// TIA Portal V18 export
// export: Created 2026-03-12T16:04:36.0251046Z, ExportSetting WithDefaults, DisplayName Totally Integrated Automation Portal, DisplayVersion V18 Update 5, DisplayName TIA Portal Openness, DisplayVersion V18 Update 5, DisplayName TIA Portal Version Control Interface, DisplayVersion V18, DisplayName SINAMICS Startdrive Advanced, DisplayVersion V18, DisplayName SINAMICS Startdrive G130, G150, S120, S150, SINAMICS MV, S210, DisplayVersion V18, DisplayName SINAMICS Startdrive G110M, G120, G120C, G120D, G120P, G115D, DisplayVersion V18, DisplayName STEP 7 Professional, DisplayVersion V18 Update 5, DisplayName STEP 7 Safety, DisplayVersion V18, DisplayName WinCC Professional, DisplayVersion V18 Update 5
FUNCTION_BLOCK "FB_MOVE_SKID_UV"   // FB40, LAD
{ S7_Optimized_Access := 'TRUE' }
VERSION : 0.1
// stored: AutoNumber true, IsIECCheckEnabled false, IsRetainMemResEnabled false, MemoryReserve 100, SetENOAutomatically false, UDAEnableTagReadback false
   VAR_INPUT
      UV_IN : Array[0..4] of Byte;
   END_VAR
   VAR_OUTPUT
      UV_OUT : Struct   // SKID Desinfecção por UV Informações monitoradas e cadastros
         LEITURA : Struct   // Endereços de Leitura (read)
            EMG_ACIONADO : Bool;   // Botão de Emergência Acionado
            REMOTO_READ : Bool;   // SKID funcionando em Modo Automático pelo nível
            "L1-1_LIGADA" : Bool;   // Status ligado/desligado Módulo de lâmpadas L1-1
            "L1-2_LIGADA" : Bool;   // Status ligado/desligado Módulo de lâmpadas L1-2
            "L1-3_LIGADA" : Bool;   // Status ligado/desligado Módulo de lâmpadas L1-3
            "L1-4_LIGADA" : Bool;   // Status ligado/desligado Módulo de lâmpadas L1-4
            "L1-5_LIGADA" : Bool;   // Status ligado/desligado Módulo de lâmpadas L1-5
            "L1-6_LIGADA" : Bool;   // Status ligado/desligado Módulo de lâmpadas L1-6
            "L1-7_LIGADA" : Bool;   // Status ligado/desligado Módulo de lâmpadas L1-7
            "L1-8_LIGADA" : Bool;   // Status ligado/desligado Módulo de lâmpadas L1-8
            "L2-1_LIGADA" : Bool;   // Status ligado/desligado Módulo de lâmpadas L2-1
            "L2-2_LIGADA" : Bool;   // Status ligado/desligado Módulo de lâmpadas L2-2
            "L2-3_LIGADA" : Bool;   // Status ligado/desligado Módulo de lâmpadas L2-3
            "L2-4_LIGADA" : Bool;   // Status ligado/desligado Módulo de lâmpadas L2-4
            "L2-5_LIGADA" : Bool;   // Status ligado/desligado Módulo de lâmpadas L2-5
            "L2-6_LIGADA" : Bool;   // Status ligado/desligado Módulo de lâmpadas L2-6
            "L2-7_LIGADA" : Bool;   // Status ligado/desligado Módulo de lâmpadas L2-7
            "L2-8_LIGADA" : Bool;   // Status ligado/desligado Módulo de lâmpadas L2-8
            "L3-1_LIGADA" : Bool;   // Status ligado/desligado Módulo de lâmpadas L3-1
            "L3-2_LIGADA" : Bool;   // Status ligado/desligado Módulo de lâmpadas L3-2
            "L3-3_LIGADA" : Bool;   // Status ligado/desligado Módulo de lâmpadas L3-3
            "L3-4_LIGADA" : Bool;   // Status ligado/desligado Módulo de lâmpadas L3-4
            "L3-5_LIGADA" : Bool;   // Status ligado/desligado Módulo de lâmpadas L3-5
            "L3-6_LIGADA" : Bool;   // Status ligado/desligado Módulo de lâmpadas L3-6
            "L3-7_LIGADA" : Bool;   // Status ligado/desligado Módulo de lâmpadas L3-7
            "L3-8_LIGADA" : Bool;   // Status ligado/desligado Módulo de lâmpadas L3-8
            "L4-1_LIGADA" : Bool;   // Status ligado/desligado Módulo de lâmpadas L4-1
            "L4-2_LIGADA" : Bool;   // Status ligado/desligado Módulo de lâmpadas L4-2
            "L4-3_LIGADA" : Bool;   // Status ligado/desligado Módulo de lâmpadas L4-3
            "L4-4_LIGADA" : Bool;   // Status ligado/desligado Módulo de lâmpadas L4-4
            "L4-5_LIGADA" : Bool;   // Status ligado/desligado Módulo de lâmpadas L4-5
            "L4-6_LIGADA" : Bool;   // Status ligado/desligado Módulo de lâmpadas L4-6
            "L4-7_LIGADA" : Bool;   // Status ligado/desligado Módulo de lâmpadas L4-7
            "L4-8_LIGADA" : Bool;   // Status ligado/desligado Módulo de lâmpadas L4-8
            RESERVA_READ_1 : Bool;   // Memória Reserva
            RESERVA_READ_2 : Bool;   // Memória Reserva
            RESERVA_READ_3 : Bool;   // Memória Reserva
            RESERVA_READ_4 : Bool;   // Memória Reserva
            RESERVA_READ_5 : Bool;   // Memória Reserva
            RESERVA_READ_6 : Bool;   // Memória Reserva
            AI1_AUX1 : DInt;   // Memória Auxiliar para escalonamento do sinal analógico do nível
            AI1_AUX2 : DInt;   // Memória Auxiliar para escalonamento do sinal analógico do nível
            NIVEL_AI1 : DInt;   // Leitura do nível aferida em metros
            "HORA_LAMP_1-1" : UInt;   // Horímetro Lâmpada 1 (Tempo em horas ligada)
            "HORA_LAMP_1-2" : UInt;   // Horímetro Lâmpada 2 (Tempo em horas ligada)
            "HORA_LAMP_1-3" : UInt;   // Horímetro Lâmpada 3 (Tempo em horas ligada)
            "HORA_LAMP_1-4" : UInt;   // Horímetro Lâmpada 4 (Tempo em horas ligada)
            "HORA_LAMP_1-5" : UInt;   // Horímetro Lâmpada 5 (Tempo em horas ligada)
            "HORA_LAMP_1-6" : UInt;   // Horímetro Lâmpada 6 (Tempo em horas ligada)
            "HORA_LAMP_1-7" : UInt;   // Horímetro Lâmpada 7 (Tempo em horas ligada)
            "HORA_LAMP_1-8" : UInt;   // Horímetro Lâmpada 8 (Tempo em horas ligada)
            "HORA_LAMP_2-1" : UInt;   // Horímetro Lâmpada 9 (Tempo em horas ligada)
            "HORA_LAMP_2-2" : UInt;   // Horímetro Lâmpada 10 (Tempo em horas ligada)
            "HORA_LAMP_2-3" : UInt;   // Horímetro Lâmpada 11 (Tempo em horas ligada)
            "HORA_LAMP_2-4" : UInt;   // Horímetro Lâmpada 12 (Tempo em horas ligada)
            "HORA_LAMP_2-5" : UInt;   // Horímetro Lâmpada 13 (Tempo em horas ligada)
            "HORA_LAMP_2-6" : UInt;   // Horímetro Lâmpada 14 (Tempo em horas ligada)
            "HORA_LAMP_2-7" : UInt;   // Horímetro Lâmpada 15 (Tempo em horas ligada)
            "HORA_LAMP_2-8" : UInt;   // Horímetro Lâmpada 16 (Tempo em horas ligada)
            "HORA_LAMP_3-1" : UInt;   // Horímetro Lâmpada 17 (Tempo em horas ligada)
            "HORA_LAMP_3-2" : UInt;   // Horímetro Lâmpada 18 (Tempo em horas ligada)
            "HORA_LAMP_3-3" : UInt;   // Horímetro Lâmpada 19 (Tempo em horas ligada)
            "HORA_LAMP_3-4" : UInt;   // Horímetro Lâmpada 20 (Tempo em horas ligada)
            "HORA_LAMP_3-5" : UInt;   // Horímetro Lâmpada 21 (Tempo em horas ligada)
            "HORA_LAMP_3-6" : UInt;   // Horímetro Lâmpada 22 (Tempo em horas ligada)
            "HORA_LAMP_3-7" : UInt;   // Horímetro Lâmpada 23 (Tempo em horas ligada)
            "HORA_LAMP_3-8" : UInt;   // Horímetro Lâmpada 24 (Tempo em horas ligada)
            "HORA_LAMP_4-1" : UInt;   // Horímetro Lâmpada 25 (Tempo em horas ligada)
            "HORA_LAMP_4-2" : UInt;   // Horímetro Lâmpada 26 (Tempo em horas ligada)
            "HORA_LAMP_4-3" : UInt;   // Horímetro Lâmpada 27 (Tempo em horas ligada)
            "HORA_LAMP_4-4" : UInt;   // Horímetro Lâmpada 28 (Tempo em horas ligada)
            "HORA_LAMP_4-5" : UInt;   // Horímetro Lâmpada 29 (Tempo em horas ligada)
            "HORA_LAMP_4-6" : UInt;   // Horímetro Lâmpada 30 (Tempo em horas ligada)
            "HORA_LAMP_4-7" : UInt;   // Horímetro Lâmpada 31 (Tempo em horas ligada)
            "HORA_LAMP_4-8" : UInt;   // Horímetro Lâmpada 32 (Tempo em horas ligada)
         END_STRUCT;
         STATUS_GERAL_1 : Bool;
         STATUS_GERAL_2 : Bool;
         STATUS_GERAL_3 : Bool;
         STATUS_GERAL_4 : Bool;   // Status para tela geral
      END_STRUCT;
   END_VAR
BEGIN

REGION Network 1: Botão de Emergência Acionado
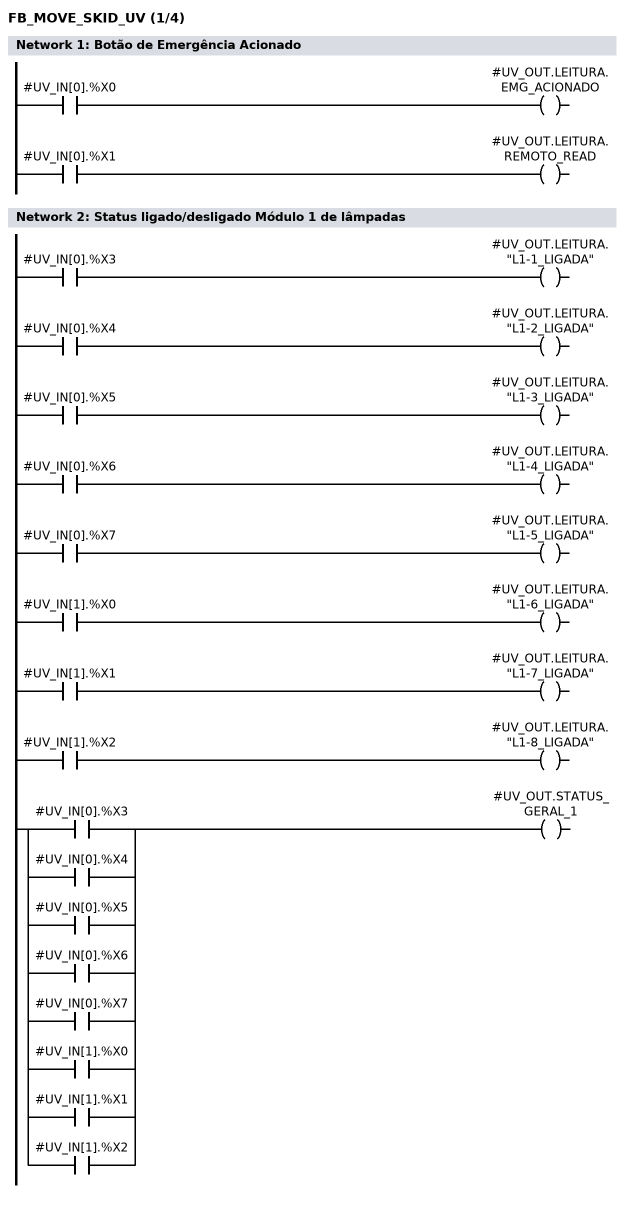
   RUNG wire#powerrail
      Contact( #UV_IN[0].%X0 )
      Coil( #UV_OUT.LEITURA.EMG_ACIONADO )
   END_RUNG
   RUNG wire#powerrail
      Contact( #UV_IN[0].%X1 )
      Coil( #UV_OUT.LEITURA.REMOTO_READ )
   END_RUNG
   // the same network as SCL:
   #UV_OUT.LEITURA.EMG_ACIONADO := #UV_IN[0].%X0;
   #UV_OUT.LEITURA.REMOTO_READ := #UV_IN[0].%X1;
END_REGION

REGION Network 2: Status ligado/desligado Módulo 1 de lâmpadas
   RUNG wire#powerrail
      Contact( #UV_IN[0].%X3 )
      Coil( #UV_OUT.LEITURA."L1-1_LIGADA" )
   END_RUNG
   RUNG wire#powerrail
      Contact( #UV_IN[0].%X4 )
      Coil( #UV_OUT.LEITURA."L1-2_LIGADA" )
   END_RUNG
   RUNG wire#powerrail
      Contact( #UV_IN[0].%X5 )
      Coil( #UV_OUT.LEITURA."L1-3_LIGADA" )
   END_RUNG
   RUNG wire#powerrail
      Contact( #UV_IN[0].%X6 )
      Coil( #UV_OUT.LEITURA."L1-4_LIGADA" )
   END_RUNG
   RUNG wire#powerrail
      Contact( #UV_IN[0].%X7 )
      Coil( #UV_OUT.LEITURA."L1-5_LIGADA" )
   END_RUNG
   RUNG wire#powerrail
      Contact( #UV_IN[1].%X0 )
      Coil( #UV_OUT.LEITURA."L1-6_LIGADA" )
   END_RUNG
   RUNG wire#powerrail
      Contact( #UV_IN[1].%X1 )
      Coil( #UV_OUT.LEITURA."L1-7_LIGADA" )
   END_RUNG
   RUNG wire#powerrail
      Contact( #UV_IN[1].%X2 )
      Coil( #UV_OUT.LEITURA."L1-8_LIGADA" )
   END_RUNG
   RUNG wire#powerrail
      Contact( #UV_IN[0].%X3 )
      wire#w1
      Coil( #UV_OUT.STATUS_GERAL_1 )
   END_RUNG
   RUNG wire#powerrail
      Contact( #UV_IN[0].%X4 )
   END_RUNG wire#w1
   RUNG wire#powerrail
      Contact( #UV_IN[0].%X5 )
   END_RUNG wire#w1
   RUNG wire#powerrail
      Contact( #UV_IN[0].%X6 )
   END_RUNG wire#w1
   RUNG wire#powerrail
      Contact( #UV_IN[0].%X7 )
   END_RUNG wire#w1
   RUNG wire#powerrail
      Contact( #UV_IN[1].%X0 )
   END_RUNG wire#w1
   RUNG wire#powerrail
      Contact( #UV_IN[1].%X1 )
   END_RUNG wire#w1
   RUNG wire#powerrail
      Contact( #UV_IN[1].%X2 )
   END_RUNG wire#w1
   // the same network as SCL:
   #UV_OUT.LEITURA."L1-1_LIGADA" := #UV_IN[0].%X3;
   #UV_OUT.LEITURA."L1-2_LIGADA" := #UV_IN[0].%X4;
   #UV_OUT.LEITURA."L1-3_LIGADA" := #UV_IN[0].%X5;
   #UV_OUT.LEITURA."L1-4_LIGADA" := #UV_IN[0].%X6;
   #UV_OUT.LEITURA."L1-5_LIGADA" := #UV_IN[0].%X7;
   #UV_OUT.LEITURA."L1-6_LIGADA" := #UV_IN[1].%X0;
   #UV_OUT.LEITURA."L1-7_LIGADA" := #UV_IN[1].%X1;
   #UV_OUT.LEITURA."L1-8_LIGADA" := #UV_IN[1].%X2;
   #UV_OUT.STATUS_GERAL_1 := #UV_IN[0].%X3 OR #UV_IN[0].%X4 OR #UV_IN[0].%X5 OR #UV_IN[0].%X6 OR #UV_IN[0].%X7 OR #UV_IN[1].%X0 OR #UV_IN[1].%X1 OR #UV_IN[1].%X2;
END_REGION

REGION Network 3: Status ligado/desligado Módulo 2 de lâmpadas
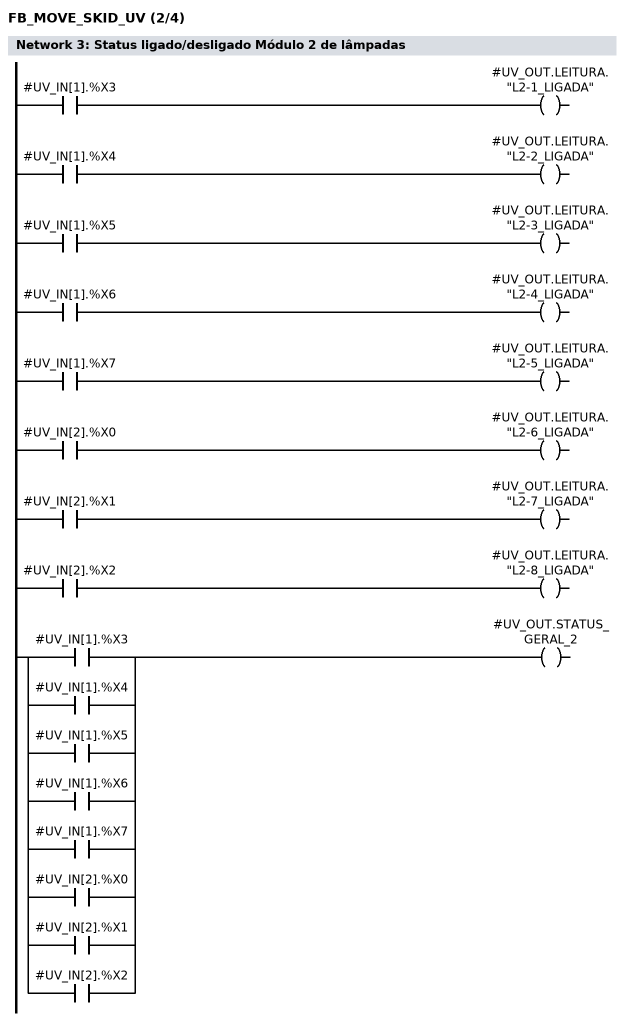
   RUNG wire#powerrail
      Contact( #UV_IN[1].%X3 )
      Coil( #UV_OUT.LEITURA."L2-1_LIGADA" )
   END_RUNG
   RUNG wire#powerrail
      Contact( #UV_IN[1].%X4 )
      Coil( #UV_OUT.LEITURA."L2-2_LIGADA" )
   END_RUNG
   RUNG wire#powerrail
      Contact( #UV_IN[1].%X5 )
      Coil( #UV_OUT.LEITURA."L2-3_LIGADA" )
   END_RUNG
   RUNG wire#powerrail
      Contact( #UV_IN[1].%X6 )
      Coil( #UV_OUT.LEITURA."L2-4_LIGADA" )
   END_RUNG
   RUNG wire#powerrail
      Contact( #UV_IN[1].%X7 )
      Coil( #UV_OUT.LEITURA."L2-5_LIGADA" )
   END_RUNG
   RUNG wire#powerrail
      Contact( #UV_IN[2].%X0 )
      Coil( #UV_OUT.LEITURA."L2-6_LIGADA" )
   END_RUNG
   RUNG wire#powerrail
      Contact( #UV_IN[2].%X1 )
      Coil( #UV_OUT.LEITURA."L2-7_LIGADA" )
   END_RUNG
   RUNG wire#powerrail
      Contact( #UV_IN[2].%X2 )
      Coil( #UV_OUT.LEITURA."L2-8_LIGADA" )
   END_RUNG
   RUNG wire#powerrail
      Contact( #UV_IN[1].%X3 )
      wire#w1
      Coil( #UV_OUT.STATUS_GERAL_2 )
   END_RUNG
   RUNG wire#powerrail
      Contact( #UV_IN[1].%X4 )
   END_RUNG wire#w1
   RUNG wire#powerrail
      Contact( #UV_IN[1].%X5 )
   END_RUNG wire#w1
   RUNG wire#powerrail
      Contact( #UV_IN[1].%X6 )
   END_RUNG wire#w1
   RUNG wire#powerrail
      Contact( #UV_IN[1].%X7 )
   END_RUNG wire#w1
   RUNG wire#powerrail
      Contact( #UV_IN[2].%X0 )
   END_RUNG wire#w1
   RUNG wire#powerrail
      Contact( #UV_IN[2].%X1 )
   END_RUNG wire#w1
   RUNG wire#powerrail
      Contact( #UV_IN[2].%X2 )
   END_RUNG wire#w1
   // the same network as SCL:
   #UV_OUT.LEITURA."L2-1_LIGADA" := #UV_IN[1].%X3;
   #UV_OUT.LEITURA."L2-2_LIGADA" := #UV_IN[1].%X4;
   #UV_OUT.LEITURA."L2-3_LIGADA" := #UV_IN[1].%X5;
   #UV_OUT.LEITURA."L2-4_LIGADA" := #UV_IN[1].%X6;
   #UV_OUT.LEITURA."L2-5_LIGADA" := #UV_IN[1].%X7;
   #UV_OUT.LEITURA."L2-6_LIGADA" := #UV_IN[2].%X0;
   #UV_OUT.LEITURA."L2-7_LIGADA" := #UV_IN[2].%X1;
   #UV_OUT.LEITURA."L2-8_LIGADA" := #UV_IN[2].%X2;
   #UV_OUT.STATUS_GERAL_2 := #UV_IN[1].%X3 OR #UV_IN[1].%X4 OR #UV_IN[1].%X5 OR #UV_IN[1].%X6 OR #UV_IN[1].%X7 OR #UV_IN[2].%X0 OR #UV_IN[2].%X1 OR #UV_IN[2].%X2;
END_REGION

REGION Network 4: Status ligado/desligado Módulo 3 de lâmpadas
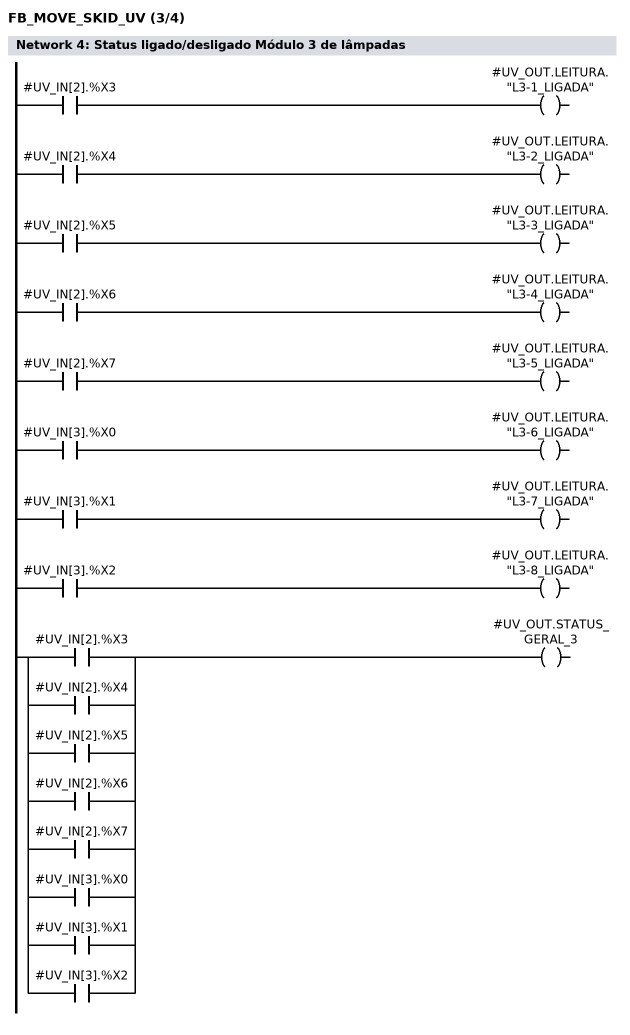
   RUNG wire#powerrail
      Contact( #UV_IN[2].%X3 )
      Coil( #UV_OUT.LEITURA."L3-1_LIGADA" )
   END_RUNG
   RUNG wire#powerrail
      Contact( #UV_IN[2].%X4 )
      Coil( #UV_OUT.LEITURA."L3-2_LIGADA" )
   END_RUNG
   RUNG wire#powerrail
      Contact( #UV_IN[2].%X5 )
      Coil( #UV_OUT.LEITURA."L3-3_LIGADA" )
   END_RUNG
   RUNG wire#powerrail
      Contact( #UV_IN[2].%X6 )
      Coil( #UV_OUT.LEITURA."L3-4_LIGADA" )
   END_RUNG
   RUNG wire#powerrail
      Contact( #UV_IN[2].%X7 )
      Coil( #UV_OUT.LEITURA."L3-5_LIGADA" )
   END_RUNG
   RUNG wire#powerrail
      Contact( #UV_IN[3].%X0 )
      Coil( #UV_OUT.LEITURA."L3-6_LIGADA" )
   END_RUNG
   RUNG wire#powerrail
      Contact( #UV_IN[3].%X1 )
      Coil( #UV_OUT.LEITURA."L3-7_LIGADA" )
   END_RUNG
   RUNG wire#powerrail
      Contact( #UV_IN[3].%X2 )
      Coil( #UV_OUT.LEITURA."L3-8_LIGADA" )
   END_RUNG
   RUNG wire#powerrail
      Contact( #UV_IN[2].%X3 )
      wire#w1
      Coil( #UV_OUT.STATUS_GERAL_3 )
   END_RUNG
   RUNG wire#powerrail
      Contact( #UV_IN[2].%X4 )
   END_RUNG wire#w1
   RUNG wire#powerrail
      Contact( #UV_IN[2].%X5 )
   END_RUNG wire#w1
   RUNG wire#powerrail
      Contact( #UV_IN[2].%X6 )
   END_RUNG wire#w1
   RUNG wire#powerrail
      Contact( #UV_IN[2].%X7 )
   END_RUNG wire#w1
   RUNG wire#powerrail
      Contact( #UV_IN[3].%X0 )
   END_RUNG wire#w1
   RUNG wire#powerrail
      Contact( #UV_IN[3].%X1 )
   END_RUNG wire#w1
   RUNG wire#powerrail
      Contact( #UV_IN[3].%X2 )
   END_RUNG wire#w1
   // the same network as SCL:
   #UV_OUT.LEITURA."L3-1_LIGADA" := #UV_IN[2].%X3;
   #UV_OUT.LEITURA."L3-2_LIGADA" := #UV_IN[2].%X4;
   #UV_OUT.LEITURA."L3-3_LIGADA" := #UV_IN[2].%X5;
   #UV_OUT.LEITURA."L3-4_LIGADA" := #UV_IN[2].%X6;
   #UV_OUT.LEITURA."L3-5_LIGADA" := #UV_IN[2].%X7;
   #UV_OUT.LEITURA."L3-6_LIGADA" := #UV_IN[3].%X0;
   #UV_OUT.LEITURA."L3-7_LIGADA" := #UV_IN[3].%X1;
   #UV_OUT.LEITURA."L3-8_LIGADA" := #UV_IN[3].%X2;
   #UV_OUT.STATUS_GERAL_3 := #UV_IN[2].%X3 OR #UV_IN[2].%X4 OR #UV_IN[2].%X5 OR #UV_IN[2].%X6 OR #UV_IN[2].%X7 OR #UV_IN[3].%X0 OR #UV_IN[3].%X1 OR #UV_IN[3].%X2;
END_REGION

REGION Network 5: Status ligado/desligado Módulo 4 de lâmpadas
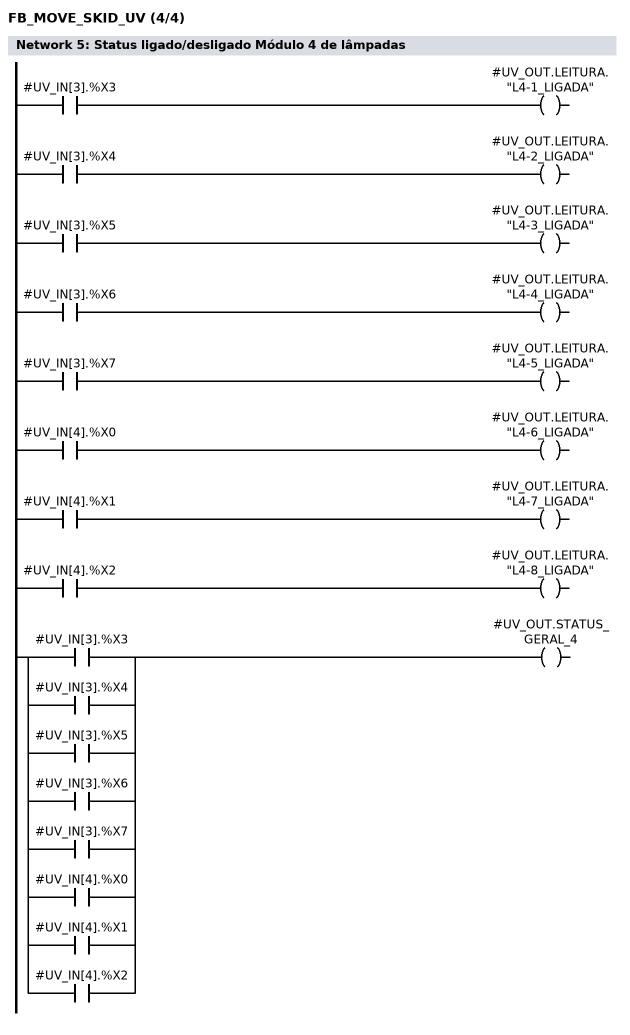
   RUNG wire#powerrail
      Contact( #UV_IN[3].%X3 )
      Coil( #UV_OUT.LEITURA."L4-1_LIGADA" )
   END_RUNG
   RUNG wire#powerrail
      Contact( #UV_IN[3].%X4 )
      Coil( #UV_OUT.LEITURA."L4-2_LIGADA" )
   END_RUNG
   RUNG wire#powerrail
      Contact( #UV_IN[3].%X5 )
      Coil( #UV_OUT.LEITURA."L4-3_LIGADA" )
   END_RUNG
   RUNG wire#powerrail
      Contact( #UV_IN[3].%X6 )
      Coil( #UV_OUT.LEITURA."L4-4_LIGADA" )
   END_RUNG
   RUNG wire#powerrail
      Contact( #UV_IN[3].%X7 )
      Coil( #UV_OUT.LEITURA."L4-5_LIGADA" )
   END_RUNG
   RUNG wire#powerrail
      Contact( #UV_IN[4].%X0 )
      Coil( #UV_OUT.LEITURA."L4-6_LIGADA" )
   END_RUNG
   RUNG wire#powerrail
      Contact( #UV_IN[4].%X1 )
      Coil( #UV_OUT.LEITURA."L4-7_LIGADA" )
   END_RUNG
   RUNG wire#powerrail
      Contact( #UV_IN[4].%X2 )
      Coil( #UV_OUT.LEITURA."L4-8_LIGADA" )
   END_RUNG
   RUNG wire#powerrail
      Contact( #UV_IN[3].%X3 )
      wire#w1
      Coil( #UV_OUT.STATUS_GERAL_4 )
   END_RUNG
   RUNG wire#powerrail
      Contact( #UV_IN[3].%X4 )
   END_RUNG wire#w1
   RUNG wire#powerrail
      Contact( #UV_IN[3].%X5 )
   END_RUNG wire#w1
   RUNG wire#powerrail
      Contact( #UV_IN[3].%X6 )
   END_RUNG wire#w1
   RUNG wire#powerrail
      Contact( #UV_IN[3].%X7 )
   END_RUNG wire#w1
   RUNG wire#powerrail
      Contact( #UV_IN[4].%X0 )
   END_RUNG wire#w1
   RUNG wire#powerrail
      Contact( #UV_IN[4].%X1 )
   END_RUNG wire#w1
   RUNG wire#powerrail
      Contact( #UV_IN[4].%X2 )
   END_RUNG wire#w1
   // the same network as SCL:
   #UV_OUT.LEITURA."L4-1_LIGADA" := #UV_IN[3].%X3;
   #UV_OUT.LEITURA."L4-2_LIGADA" := #UV_IN[3].%X4;
   #UV_OUT.LEITURA."L4-3_LIGADA" := #UV_IN[3].%X5;
   #UV_OUT.LEITURA."L4-4_LIGADA" := #UV_IN[3].%X6;
   #UV_OUT.LEITURA."L4-5_LIGADA" := #UV_IN[3].%X7;
   #UV_OUT.LEITURA."L4-6_LIGADA" := #UV_IN[4].%X0;
   #UV_OUT.LEITURA."L4-7_LIGADA" := #UV_IN[4].%X1;
   #UV_OUT.LEITURA."L4-8_LIGADA" := #UV_IN[4].%X2;
   #UV_OUT.STATUS_GERAL_4 := #UV_IN[3].%X3 OR #UV_IN[3].%X4 OR #UV_IN[3].%X5 OR #UV_IN[3].%X6 OR #UV_IN[3].%X7 OR #UV_IN[4].%X0 OR #UV_IN[4].%X1 OR #UV_IN[4].%X2;
END_REGION
END_FUNCTION_BLOCK
